// TwinCAT 3 PLC project Core
// Title: Twincat Open Library
// Company: Home
// ProjectVersion: 1.0.0.4
// ProgramVersion: 3.1.4026.17
// libraries:
//   Tc2_Standard, * (Beckhoff Automation GmbH)
//   Tc2_System, * (Beckhoff Automation GmbH)
//   Tc3_Module, * (Beckhoff Automation GmbH)
// project tree:
//   Modules/Common/ E_Requester.TcDUT (not stored), E_RpcMethodResponse.TcDUT, F_ValidateRequester.TcPOU (not stored)
//   Modules/Pneumatics/TwoPosActuator/ E_TwoPosActuator_Fault.TcDUT (not stored), E_TwoPosActuator_State.TcDUT (not stored), FB_TwoPosActuator.TcPOU, ST_TwoPosActuator_Cfg.TcDUT (not stored), ST_TwoPosActuator_IO.TcDUT (not stored), ST_TwoPosActuator_Sts.TcDUT (not stored)
//   Modules/Interlocks/ FB_Interlock.TcPOU (not stored), ST_Interlock_Config.TcDUT (not stored), ST_Interlock_Status.TcDUT (not stored), ST_Interlock_Faceplate.TcDUT (not stored)
//   Modules/Sequencing/Permissives/ FB_Permissives.TcPOU, ST_Permissive_Config.TcDUT (not stored), ST_Permissive_Status.TcDUT (not stored), ST_Permissive_Faceplate.TcDUT
//   Modules/Sequencing/StateMachine/ E_SM_State.TcDUT, FB_StateMachine.TcPOU, FB_Step.TcPOU, ST_SM_Status.TcDUT, ST_SM_Step.TcDUT
//   / PlcTask.TcTTO (not stored)
// (motion and I/O tree: see PLC project coreexample)
// real-time tasks:
//   TASK PlcTask: cycle T#10ms, priority 20, ADS port 350
//   TASK VISU_TASK: cycle T#200000us, priority 30, ADS port 351
//   TASK IO Task New: cycle T#1ms, priority 1, ADS port 301
// variable links:

// ---- Modules/Common/E_RpcMethodResponse.TcDUT
{attribute 'qualified_only'}
{attribute 'strict'}
{attribute 'to_string'}
TYPE E_RpcMethodResponse :
(
    // Success (0)
    ACCEPTED := 0,
    
    // Source / Authorization (10-19)
    REJECTED_SOURCE_NOT_ALLOWED := 11,
    
    // State rejection (20-29)
    REJECTED_WRONG_STATE := 20,
    REJECTED_FAULTED := 21,
    REJECTED_ALREADY_AT_TARGET := 23,
    
    // Parameter / Config (30-39)
    REJECTED_INVALID_PARAMETER := 30,
    REJECTED_BYPASS_NOT_ALLOWED := 31,
    
    // Permissive / Interlock (50-59)
    REJECTED_PERMISSIVE_NOT_MET := 50,
    REJECTED_INTERLOCKED := 51,
    
    // Default (100)
    REJECTED_UNKNOWN := 100
);
END_TYPE

// ---- Modules/Sequencing/Permissives/ST_Permissive_Faceplate.TcDUT
(*
Permissive Faceplate Structure
==============================
Individual permissive bit information for HMI faceplate display
*)
{attribute 'OPC.UA.DA' := '1'}
{attribute 'OPC.UA.DA.Access' := '1'}
{attribute 'OPC.UA.DA.StructuredType' := '1'}
TYPE ST_Permissive_Faceplate :
STRUCT
	{attribute 'OPC.UA.DA.Description' := 'Human readable name of the permissive'}
	name : STRING(50);
	{attribute 'OPC.UA.DA.Description' := 'Real-time status of this permissive bit (TRUE=good, FALSE=bad)'}
	stsOK : BOOL;
	{attribute 'OPC.UA.DA.Description' := 'TRUE if this bit is actively mapped via MapInput'}
	stsMapped : BOOL;
	{attribute 'OPC.UA.DA.Description' := 'TRUE if this bit is currently bypassed'}
	stsBypassed : BOOL;
	{attribute 'OPC.UA.DA.Description' := 'TRUE if this bit is configured as bypassable'}
	cfgBypassable : BOOL;
END_STRUCT
END_TYPE

// ---- Modules/Sequencing/StateMachine/E_SM_State.TcDUT
{attribute 'qualified_only'}
{attribute 'strict'}
{attribute 'to_string'}
TYPE E_SM_State :
(
    IDLE        := 0,
    RUNNING     := 1,
    STOPPING    := 2,
    HOMING      := 4,
    ABORTING    := 8,
    HOMED       := 16,
    STOPPED     := 32,
    ABORTED     := 64,
    COMPLETE    := 128,
    PAUSING     := 256,
    PAUSED      := 512,
    PROCEEDING  := 1024
);
END_TYPE

// ---- Modules/Sequencing/StateMachine/ST_SM_Status.TcDUT
TYPE ST_SM_Status :
STRUCT
    // Current state (enum with to_string for HMI)
    State : E_SM_State := E_SM_State.STOPPED;
    LastState : E_SM_State := E_SM_State.STOPPED;
    
    // Derived state categories
    ActiveState : BOOL;
    WaitingState : BOOL;
    
    // Computed status
    Faulted : BOOL;
    SubmoduleFaulted : BOOL;
    Blocked : BOOL;
    Starved : BOOL;
    
    // Permission-derived readiness
    ReadyToHome : BOOL;
    ReadyToStart : BOOL;
    ReadyToProceed : BOOL;
    
    // Auto-run tracking
    AutoStartRequest : BOOL;
    AutoCycleRequest : BOOL;
END_STRUCT
END_TYPE

// ---- Modules/Sequencing/StateMachine/ST_SM_Step.TcDUT
(*
Active step snapshot published by FB_StateMachine.
FB_Step writes the name and permissives into here while it is the
active step. Number, next target, and timer are owned by the state
machine itself.
*)
{attribute 'OPC.UA.DA' := '1'}
{attribute 'OPC.UA.DA.Access' := '1'}
{attribute 'OPC.UA.DA.StructuredType' := '1'}
TYPE ST_SM_Step :
STRUCT
    {attribute 'OPC.UA.DA.Description' := 'Active step number'}
    Current : DINT;

    {attribute 'OPC.UA.DA.Description' := 'Active step name (published by FB_Step)'}
    Name : STRING(40);

    {attribute 'OPC.UA.DA.Description' := 'Step the state machine will transition to next'}
    Next : DINT;

    {attribute 'OPC.UA.DA.Description' := 'Seconds spent in the active step'}
    TimerSeconds : REAL;

    {attribute 'OPC.UA.DA.Description' := 'Config of the active step permissives'}
    PermCfg : ST_Permissive_Config;

    {attribute 'OPC.UA.DA.Description' := 'Status of the active step permissives'}
    PermStatus : ST_Permissive_Status;
END_STRUCT
END_TYPE

// ---- Modules/Pneumatics/TwoPosActuator/FB_TwoPosActuator.TcPOU
{attribute 'OPC.UA.DA' := '1'}
FUNCTION_BLOCK FB_TwoPosActuator
VAR_INPUT
    {attribute 'OPC.UA.DA' := '0'}
    EnableIn : BOOL := TRUE;
    
    // Configuration
    {attribute 'OPC.UA.DA' := '1'}
    {attribute 'OPC.UA.DA.Access' := '1'}
    cfg : ST_TwoPosActuator_Cfg;
END_VAR

VAR_OUTPUT
    {attribute 'OPC.UA.DA' := '0'}
    EnableOut : BOOL;
    {attribute 'OPC.UA.DA' := '1'}
    {attribute 'OPC.UA.DA.Access' := '1'}
    sts : ST_TwoPosActuator_Sts;
END_VAR

VAR_IN_OUT
    {attribute 'OPC.UA.DA' := '0'}
    IO : ST_TwoPosActuator_IO;
END_VAR

VAR
    // Composed modules - permissive handlers (visible on OPC)
    advancePermissives : FB_Permissives;
    retractPermissives : FB_Permissives;
    
    // Internal state machine
    {attribute 'OPC.UA.DA' := '0'}
    currentState : E_TwoPosActuator_State := E_TwoPosActuator_State.Undefined;
    {attribute 'OPC.UA.DA' := '0'}
    previousState : E_TwoPosActuator_State;
    
    // Timers for motion
    {attribute 'OPC.UA.DA' := '0'}
    advanceTimer : TON;
    {attribute 'OPC.UA.DA' := '0'}
    retractTimer : TON;
    
    // Edge detection
    {attribute 'OPC.UA.DA' := '0'}
    rTrigAdvanced : R_TRIG;
    {attribute 'OPC.UA.DA' := '0'}
    rTrigRetracted : R_TRIG;
    
    // Internal flags
    {attribute 'OPC.UA.DA' := '0'}
    bothFeedbackActive : BOOL;
    
    // Fault handling
    {attribute 'OPC.UA.DA' := '0'}
    faultLatched : BOOL;
    {attribute 'OPC.UA.DA' := '0'}
    lastFault : E_TwoPosActuator_Fault;
    {attribute 'OPC.UA.DA' := '0'}
    bSourceLockedToProg : BOOL;
END_VAR

//-----------------------------------------------------------------------------
// Main Implementation - FB_TwoPosActuator
// Cyclic monitoring only. All commands issued via methods.
//-----------------------------------------------------------------------------
EnableOut := EnableIn;

IF EnableIn THEN
    
    //-------------------------------------------------------------------------
    // Permissive Evaluation
    //-------------------------------------------------------------------------
    advancePermissives();
    retractPermissives();
    
    //-------------------------------------------------------------------------
    // Feedback Analysis
    //-------------------------------------------------------------------------
    bothFeedbackActive := IO.inFbkAdvanced AND IO.inFbkRetracted;
    
    //-------------------------------------------------------------------------
    // State Machine - Cyclic Monitoring
    // Methods set currentState and IO; body monitors for completion/faults.
    //-------------------------------------------------------------------------
    previousState := currentState;
    
    CASE currentState OF
        
        E_TwoPosActuator_State.Undefined:
            IO.outValveAdvance := FALSE;
            IO.outValveRetract := FALSE;
            
            IF bothFeedbackActive THEN
                currentState := E_TwoPosActuator_State.Fault;
                sts.faultCode := E_TwoPosActuator_Fault.BothFeedbackOn;
                faultLatched := TRUE;
            ELSIF IO.inFbkAdvanced AND NOT IO.inFbkRetracted THEN
                currentState := E_TwoPosActuator_State.Advanced;
            ELSIF IO.inFbkRetracted AND NOT IO.inFbkAdvanced THEN
                currentState := E_TwoPosActuator_State.Retracted;
            END_IF;
        
        E_TwoPosActuator_State.Retracted:
            IF cfg.cfgHoldAtRetracted THEN
                IO.outValveRetract := TRUE;
            ELSE
                IO.outValveRetract := FALSE;
            END_IF;
            IO.outValveAdvance := FALSE;
            
            IF bothFeedbackActive THEN
                currentState := E_TwoPosActuator_State.Fault;
                sts.faultCode := E_TwoPosActuator_Fault.BothFeedbackOn;
                faultLatched := TRUE;
            ELSIF NOT IO.inFbkRetracted THEN
                currentState := E_TwoPosActuator_State.Fault;
                sts.faultCode := E_TwoPosActuator_Fault.UndefinedState;
                faultLatched := TRUE;
            END_IF;
        
        E_TwoPosActuator_State.Advancing:
            IO.outValveAdvance := TRUE;
            IO.outValveRetract := FALSE;
            advanceTimer(IN := TRUE, PT := DINT_TO_TIME(cfg.cfgAdvTimeoutS * 1000));
            
            IF IO.inFbkAdvanced AND NOT IO.inFbkRetracted THEN
                currentState := E_TwoPosActuator_State.Advanced;
                advanceTimer(IN := FALSE);
            ELSIF advanceTimer.Q THEN
                currentState := E_TwoPosActuator_State.Fault;
                sts.faultCode := E_TwoPosActuator_Fault.AdvanceTimeout;
                faultLatched := TRUE;
                advanceTimer(IN := FALSE);
            ELSIF bothFeedbackActive THEN
                currentState := E_TwoPosActuator_State.Fault;
                sts.faultCode := E_TwoPosActuator_Fault.BothFeedbackOn;
                faultLatched := TRUE;
                advanceTimer(IN := FALSE);
            ELSIF NOT advancePermissives.sts.bOK THEN
                currentState := E_TwoPosActuator_State.Fault;
                sts.faultCode := E_TwoPosActuator_Fault.PermissivesNotOK;
                faultLatched := TRUE;
                advanceTimer(IN := FALSE);
            END_IF;
        
        E_TwoPosActuator_State.Advanced:
            IF cfg.cfgHoldAtAdvanced THEN
                IO.outValveAdvance := TRUE;
            ELSE
                IO.outValveAdvance := FALSE;
            END_IF;
            IO.outValveRetract := FALSE;
            
            IF bothFeedbackActive THEN
                currentState := E_TwoPosActuator_State.Fault;
                sts.faultCode := E_TwoPosActuator_Fault.BothFeedbackOn;
                faultLatched := TRUE;
            ELSIF NOT IO.inFbkAdvanced THEN
                currentState := E_TwoPosActuator_State.Fault;
                sts.faultCode := E_TwoPosActuator_Fault.UndefinedState;
                faultLatched := TRUE;
            END_IF;
        
        E_TwoPosActuator_State.Retracting:
            IO.outValveRetract := TRUE;
            IO.outValveAdvance := FALSE;
            retractTimer(IN := TRUE, PT := DINT_TO_TIME(cfg.cfgRetTimeoutS * 1000));
            
            IF IO.inFbkRetracted AND NOT IO.inFbkAdvanced THEN
                currentState := E_TwoPosActuator_State.Retracted;
                retractTimer(IN := FALSE);
            ELSIF retractTimer.Q THEN
                currentState := E_TwoPosActuator_State.Fault;
                sts.faultCode := E_TwoPosActuator_Fault.RetractTimeout;
                faultLatched := TRUE;
                retractTimer(IN := FALSE);
            ELSIF bothFeedbackActive THEN
                currentState := E_TwoPosActuator_State.Fault;
                sts.faultCode := E_TwoPosActuator_Fault.BothFeedbackOn;
                faultLatched := TRUE;
                retractTimer(IN := FALSE);
            ELSIF NOT retractPermissives.sts.bOK THEN
                currentState := E_TwoPosActuator_State.Fault;
                sts.faultCode := E_TwoPosActuator_Fault.PermissivesNotOK;
                faultLatched := TRUE;
                retractTimer(IN := FALSE);
            END_IF;
        
        E_TwoPosActuator_State.Fault:
            IO.outValveAdvance := FALSE;
            IO.outValveRetract := FALSE;
            advanceTimer(IN := FALSE);
            retractTimer(IN := FALSE);
    END_CASE;
    
    //-------------------------------------------------------------------------
    // Status Output Generation
    //-------------------------------------------------------------------------
    sts.state := currentState;
    sts.stsAdvanced := (currentState = E_TwoPosActuator_State.Advanced);
    sts.stsRetracted := (currentState = E_TwoPosActuator_State.Retracted);
    sts.stsMoving := (currentState = E_TwoPosActuator_State.Advancing) OR 
                     (currentState = E_TwoPosActuator_State.Retracting);
    sts.stsFaulted := (currentState = E_TwoPosActuator_State.Fault) OR faultLatched;
    sts.lastFaultCode := lastFault;
    
    rTrigAdvanced(CLK := sts.stsAdvanced);
    sts.osAdvanced := rTrigAdvanced.Q;
    
    rTrigRetracted(CLK := sts.stsRetracted);
    sts.osRetracted := rTrigRetracted.Q;
    
    //-------------------------------------------------------------------------
    // String Generation for OPC/HMI
    //-------------------------------------------------------------------------
    CASE currentState OF
        E_TwoPosActuator_State.Undefined:   sts.stateString := 'Undefined';
        E_TwoPosActuator_State.Retracted:   sts.stateString := 'Retracted';
        E_TwoPosActuator_State.Advancing:   sts.stateString := 'Advancing';
        E_TwoPosActuator_State.Advanced:    sts.stateString := 'Advanced';
        E_TwoPosActuator_State.Retracting:  sts.stateString := 'Retracting';
        E_TwoPosActuator_State.Fault:       sts.stateString := 'Fault';
    ELSE
        sts.stateString := 'Unknown';
    END_CASE;
    
    CASE sts.faultCode OF
        E_TwoPosActuator_Fault.None:               sts.faultString := 'No Fault';
        E_TwoPosActuator_Fault.AdvanceTimeout:      sts.faultString := 'Advance Timeout';
        E_TwoPosActuator_Fault.RetractTimeout:      sts.faultString := 'Retract Timeout';
        E_TwoPosActuator_Fault.BothFeedbackOn:      sts.faultString := 'Both Feedbacks Active';
        E_TwoPosActuator_Fault.UndefinedState:      sts.faultString := 'Position Undefined';
        E_TwoPosActuator_Fault.PermissivesNotOK:    sts.faultString := 'Permissives Not OK';
        E_TwoPosActuator_Fault.ConflictingCommands:  sts.faultString := 'Conflicting Commands';
        E_TwoPosActuator_Fault.NoFeedback:          sts.faultString := 'No Position Feedback';
    ELSE
        sts.faultString := 'Unknown Fault';
    END_CASE;
    
    CASE sts.lastFaultCode OF
        E_TwoPosActuator_Fault.None:               sts.lastFaultString := 'No Previous Fault';
        E_TwoPosActuator_Fault.AdvanceTimeout:      sts.lastFaultString := 'Last: Advance Timeout';
        E_TwoPosActuator_Fault.RetractTimeout:      sts.lastFaultString := 'Last: Retract Timeout';
        E_TwoPosActuator_Fault.BothFeedbackOn:      sts.lastFaultString := 'Last: Both Feedbacks Active';
        E_TwoPosActuator_Fault.UndefinedState:      sts.lastFaultString := 'Last: Position Undefined';
        E_TwoPosActuator_Fault.PermissivesNotOK:    sts.lastFaultString := 'Last: Permissives Not OK';
        E_TwoPosActuator_Fault.ConflictingCommands:  sts.lastFaultString := 'Last: Conflicting Commands';
        E_TwoPosActuator_Fault.NoFeedback:          sts.lastFaultString := 'Last: No Position Feedback';
    ELSE
        sts.lastFaultString := 'Last: Unknown Fault';
    END_CASE;
    
ELSE
    IO.outValveAdvance := FALSE;
    IO.outValveRetract := FALSE;
    advanceTimer(IN := FALSE);
    retractTimer(IN := FALSE);
END_IF;

{attribute 'TcRpcEnable' := '1'}
METHOD PUBLIC Advance : E_RpcMethodResponse
VAR_INPUT
    eRequester : E_Requester := E_Requester.PROG;
END_VAR
// 1. Source + fault validation
Advance := F_ValidateRequester(eRequester, bSourceLockedToProg, faultLatched, FALSE, FALSE);
IF Advance <> E_RpcMethodResponse.ACCEPTED THEN RETURN; END_IF;

// 2. State check — must not already be advanced or advancing
IF currentState = E_TwoPosActuator_State.Advanced OR currentState = E_TwoPosActuator_State.Advancing THEN
    Advance := E_RpcMethodResponse.REJECTED_ALREADY_AT_TARGET;
    RETURN;
END_IF;

// 3. Permissive check
IF NOT advancePermissives.sts.bOK THEN
    Advance := E_RpcMethodResponse.REJECTED_PERMISSIVE_NOT_MET;
    RETURN;
END_IF;

// 4. Execute — set state, body handles the rest
currentState := E_TwoPosActuator_State.Advancing;
advanceTimer(IN := FALSE);
Advance := E_RpcMethodResponse.ACCEPTED;
END_METHOD

{attribute 'TcRpcEnable' := '1'}
METHOD PUBLIC Retract : E_RpcMethodResponse
VAR_INPUT
    eRequester : E_Requester := E_Requester.PROG;
END_VAR
// 1. Source + fault validation
Retract := F_ValidateRequester(eRequester, bSourceLockedToProg, faultLatched, FALSE, FALSE);
IF Retract <> E_RpcMethodResponse.ACCEPTED THEN RETURN; END_IF;

// 2. State check — must not already be retracted or retracting
IF currentState = E_TwoPosActuator_State.Retracted OR currentState = E_TwoPosActuator_State.Retracting THEN
    Retract := E_RpcMethodResponse.REJECTED_ALREADY_AT_TARGET;
    RETURN;
END_IF;

// 3. Permissive check
IF NOT retractPermissives.sts.bOK THEN
    Retract := E_RpcMethodResponse.REJECTED_PERMISSIVE_NOT_MET;
    RETURN;
END_IF;

// 4. Execute — set state, body handles the rest
currentState := E_TwoPosActuator_State.Retracting;
retractTimer(IN := FALSE);
Retract := E_RpcMethodResponse.ACCEPTED;
END_METHOD

{attribute 'TcRpcEnable' := '1'}
METHOD PUBLIC AllOff : E_RpcMethodResponse
VAR_INPUT
    eRequester : E_Requester := E_Requester.PROG;
END_VAR
// AllOff is always accepted — safety command
AllOff := F_ValidateRequester(eRequester, bSourceLockedToProg, faultLatched, FALSE, TRUE);
IF AllOff <> E_RpcMethodResponse.ACCEPTED THEN RETURN; END_IF;

IO.outValveAdvance := FALSE;
IO.outValveRetract := FALSE;
advanceTimer(IN := FALSE);
retractTimer(IN := FALSE);
currentState := E_TwoPosActuator_State.Undefined;
AllOff := E_RpcMethodResponse.ACCEPTED;
END_METHOD

{attribute 'TcRpcEnable' := '1'}
METHOD PUBLIC Reset : E_RpcMethodResponse
VAR_INPUT
    eRequester : E_Requester := E_Requester.PROG;
END_VAR
// 1. Source validation — allow when faulted
Reset := F_ValidateRequester(eRequester, bSourceLockedToProg, faultLatched, TRUE, FALSE);
IF Reset <> E_RpcMethodResponse.ACCEPTED THEN RETURN; END_IF;

// 2. Must be in fault state
IF currentState <> E_TwoPosActuator_State.Fault THEN
    Reset := E_RpcMethodResponse.REJECTED_WRONG_STATE;
    RETURN;
END_IF;

// 3. Execute — clear fault and go to Undefined for re-evaluation
lastFault := sts.faultCode;
faultLatched := FALSE;
sts.faultCode := E_TwoPosActuator_Fault.None;
currentState := E_TwoPosActuator_State.Undefined;
IO.outValveAdvance := FALSE;
IO.outValveRetract := FALSE;
Reset := E_RpcMethodResponse.ACCEPTED;
END_METHOD

{attribute 'TcRpcEnable' := '1'}
METHOD PUBLIC LockSource : E_RpcMethodResponse
VAR_INPUT
    bLock : BOOL;
END_VAR
bSourceLockedToProg := bLock;
LockSource := E_RpcMethodResponse.ACCEPTED;
END_METHOD

END_FUNCTION_BLOCK

// ---- Modules/Sequencing/Permissives/FB_Permissives.TcPOU
(*
PERMISSIVE - Operational Enabling Function Block
================================================
Philosophy: 	Allows a change in state when all conditions are met
Behavior: 		Follows real-time conditions, no latching, can be bypassed for maintenance
Logic: 			Mapped bits: 1 = good, 0 = bad. Unmapped bits are automatically good (1)
				sts.bOK = TRUE when ALL active permissive bits are good (or bypassed)
				Non-latching - immediate response to condition changes
Mapping:		Use MapInput method to assign boolean signals to specific bits (0..63)
				Unmapped bits automatically return to good state after timeout
*)
{attribute 'OPC.UA.DA' := '1'}
FUNCTION_BLOCK PUBLIC FB_Permissives
VAR_INPUT
	{attribute 'OPC.UA.DA' := '1'}
	{attribute 'OPC.UA.DA.Access' := '1'}
	cfg : ST_Permissive_Config;
END_VAR
VAR_OUTPUT
	{attribute 'OPC.UA.DA' := '1'}
	{attribute 'OPC.UA.DA.Access' := '1'}
	sts : ST_Permissive_Status;
END_VAR
VAR
	{attribute 'OPC.UA.DA' := '0'}
	_permissiveBits : ULINT := 16#FFFFFFFFFFFFFFFF;	// Working bits (1=good, 0=bad), default all good
	{attribute 'OPC.UA.DA' := '0'}
	_activeMask : ULINT := 0;							// Tracks which bits are actively mapped
	{attribute 'OPC.UA.DA' := '0'}
	_bypassMask : ULINT := 0;							// Dynamic bypass mask (1=bypassed)
	{attribute 'OPC.UA.DA' := '0'}
	_previousBits : ULINT := 16#FFFFFFFFFFFFFFFF;		// Previous cycle bits for transition detection
	{attribute 'OPC.UA.DA' := '0'}
	_cycleCounter : UDINT := 0;
	{attribute 'OPC.UA.DA' := '0'}
	_lastMappedCycle : ARRAY[0..63] OF UDINT;
	{attribute 'OPC.UA.DA' := '0'}
	_sequenceCounter : UDINT := 0;
	{attribute 'OPC.UA.DA' := '0'}
	MAPPING_TIMEOUT : UDINT := 10;						// Cycles before considering a bit unmapped
END_VAR

// Increment cycle counter
_cycleCounter := _cycleCounter + 1;
IF _cycleCounter = 0 THEN _cycleCounter := 1; END_IF

// Cleanup unmapped bits
CleanupUnmappedBits();

// Detect transitions for first-failure tracking
DetectTransitions();

// Compute permissive status: unmapped bits default good, then apply bypass
sts.nPermissives := (_permissiveBits OR NOT _activeMask) OR _bypassMask;
sts.nBypassMask := _bypassMask;

// Overall OK: all 64 bits good
sts.bOK := sts.nPermissives = 16#FFFFFFFFFFFFFFFF;

// Update faceplates for HMI
UpdateFaceplates();

// Store for next cycle transition detection
_previousBits := _permissiveBits;

METHOD PRIVATE CleanupUnmappedBits
VAR
	i : UDINT;
	bitMask : ULINT;
END_VAR
FOR i := 0 TO 63 DO
	bitMask := SHL(ULINT#1, i);
	IF (_activeMask AND bitMask) <> 0 THEN
		IF (_cycleCounter - _lastMappedCycle[i]) > MAPPING_TIMEOUT THEN
			_activeMask := _activeMask AND NOT bitMask;
			_permissiveBits := _permissiveBits OR bitMask;	// Reset to good
		END_IF
	END_IF
END_FOR;
END_METHOD

METHOD PRIVATE DetectTransitions
VAR
	i : UDINT;
	bitMask : ULINT;
END_VAR
// New failure sequence: transition from all-good to first failure
IF _previousBits = 16#FFFFFFFFFFFFFFFF AND _permissiveBits <> 16#FFFFFFFFFFFFFFFF THEN
	_sequenceCounter := 0;
	sts.nFirstFailureBitIndex := 999;
END_IF

// Detect good-to-bad transitions on active bits
FOR i := 0 TO 63 DO
	bitMask := SHL(ULINT#1, i);
	IF (_activeMask AND bitMask) <> 0 THEN
		// Previous good (1) AND current bad (0) = transition
		IF ((_previousBits AND bitMask) <> 0) AND ((_permissiveBits AND bitMask) = 0) THEN
			_sequenceCounter := _sequenceCounter + 1;
			IF _sequenceCounter = 1 THEN
				sts.nFirstFailureBitIndex := i;
			END_IF
		END_IF
	END_IF
END_FOR;
END_METHOD

(*
Map a boolean input signal to a specific permissive bit (0..63)
Call every cycle for each active permissive condition
*)
METHOD PUBLIC MapInput
VAR_INPUT
	bitIndex : UDINT;
	inputValue : BOOL;
END_VAR
VAR
	bitMask : ULINT;
END_VAR
IF bitIndex > 63 THEN RETURN; END_IF

bitMask := SHL(ULINT#1, bitIndex);
_activeMask := _activeMask OR bitMask;
_lastMappedCycle[bitIndex] := _cycleCounter;

IF inputValue THEN
	_permissiveBits := _permissiveBits OR bitMask;
ELSE
	_permissiveBits := _permissiveBits AND NOT bitMask;
END_IF;
END_METHOD

(*
Reset - Clear all bypass states
Permissives continue to follow real-time conditions (non-latching)
*)
{attribute 'TcRpcEnable':='1'}
METHOD Reset
_bypassMask := 0;
END_METHOD

(*
Set or clear bypass for a specific permissive bit
Only bits configured as bypassable in cfg.nBypassable can be bypassed
Clearing bypass (bEnable := FALSE) is always allowed
*)
{attribute 'TcRpcEnable':='1'}
METHOD PUBLIC SetBypass : E_RpcMethodResponse
VAR_INPUT
	bitIndex : UDINT;
	bEnable : BOOL;
END_VAR
VAR
	bitMask : ULINT;
END_VAR
IF bitIndex > 63 THEN
	SetBypass := E_RpcMethodResponse.REJECTED_INVALID_PARAMETER;
	RETURN;
END_IF

bitMask := SHL(ULINT#1, bitIndex);

// Only check bypassable config when enabling
IF bEnable AND (cfg.nBypassable AND bitMask) = 0 THEN
	SetBypass := E_RpcMethodResponse.REJECTED_BYPASS_NOT_ALLOWED;
	RETURN;
END_IF

IF bEnable THEN
	_bypassMask := _bypassMask OR bitMask;
ELSE
	_bypassMask := _bypassMask AND NOT bitMask;
END_IF

SetBypass := E_RpcMethodResponse.ACCEPTED;
END_METHOD

METHOD PRIVATE UpdateFaceplates
VAR
	i : UDINT;
	bitMask : ULINT;
END_VAR
FOR i := 0 TO 63 DO
	bitMask := SHL(ULINT#1, i);
	sts.aFaceplates[i].name := cfg.aNames[i];
	sts.aFaceplates[i].stsOK := (sts.nPermissives AND bitMask) <> 0;
	sts.aFaceplates[i].stsMapped := (_activeMask AND bitMask) <> 0;
	sts.aFaceplates[i].stsBypassed := (_bypassMask AND bitMask) <> 0;
	sts.aFaceplates[i].cfgBypassable := (cfg.nBypassable AND bitMask) <> 0;
END_FOR;
END_METHOD

END_FUNCTION_BLOCK

// ---- Modules/Sequencing/StateMachine/FB_StateMachine.TcPOU
FUNCTION_BLOCK FB_StateMachine
VAR_INPUT
    EnableIn : BOOL;
    cfgAutoRun : BOOL;
    inpBlockedCondition : DINT;
    inpStarvedCondition : DINT;
    inpSubmoduleFaulted : BOOL;
END_VAR

VAR_OUTPUT
    EnableOut : BOOL;
    Status : ST_SM_Status;
END_VAR

VAR CONSTANT
    HOMING_MIN   : DINT := 1000; HOMING_MAX   : DINT := 1999;
    RUNNING_MIN  : DINT := 3000; RUNNING_MAX  : DINT := 3999;
    STOPPING_MIN : DINT := 2000; STOPPING_MAX : DINT := 2999;
    ABORTING_MIN : DINT := 5000; ABORTING_MAX : DINT := 5999;
    PAUSING_MIN  : DINT := 4000; PAUSING_MAX  : DINT := 4999;
    PROCEEDING_MIN : DINT := 6000; PROCEEDING_MAX : DINT := 6999;
END_VAR

VAR
    // Internal command request flags (set by methods, consumed by body)
    _abortRequested : BOOL;
    _completeStateRequested : BOOL;
    _homeRequested : BOOL;
    _pauseRequested : BOOL;
    _proceedRequested : BOOL;
    _startRequested : BOOL;
    _stopRequested : BOOL;
    _retryActive : BOOL;
    RetryComplete : BOOL;
    
    // Timer
    StepTimer : TON;
    
    // Edge detection
    R_TRIG_1 : R_TRIG;
    R_TRIG_5 : R_TRIG;
    
    // Internal state tracking
    _previousState : E_SM_State;
    PreviousStep : DINT;
    TimerReset : BOOL;
    LsOdd : DINT;
    _returnState : E_SM_State;
    ReturnNextStep : DINT;
    
    // Permission handlers
    permAuto : FB_Permissives;
    permHome : FB_Permissives;
    permProceed : FB_Permissives;
    permStart : FB_Permissives;
    
    // Running interlock (latching - auto-aborts from any active state)
    intlkRunning : FB_Interlock;
    
    // Temp variables
    permIndex : UDINT;
    stepIsZero : BOOL;
    seqDone : BOOL;
    
    // Source control
    bSourceLockedToProg : BOOL;
    
    // Step ownership (internal)
    _nextStep : DINT;
END_VAR


//-----------------------------------------------------------------------------
// Main Implementation
//-----------------------------------------------------------------------------
EnableOut := EnableIn;

// Only execute if enabled
IF EnableIn THEN
    //-------------------------------------------------------------------------
    // Process permissions for different states
    //-------------------------------------------------------------------------
    permHome();
    permStart();
    permProceed();
    permAuto();
    
    intlkRunning();
    
    // Auto-abort if any running interlock trips (e-stop, safety gate, etc.)
    IF NOT intlkRunning.sts.bOK AND
       NOT (Status.State = E_SM_State.STOPPED OR Status.State = E_SM_State.ABORTING) THEN
        _abortRequested := TRUE;
    END_IF;
    
    //-------------------------------------------------------------------------
    // Ready state calculations
    //-------------------------------------------------------------------------
    Status.ReadyToHome := (Status.State = E_SM_State.STOPPED) AND
                          permHome.sts.bOK AND
                          permAuto.sts.bOK;

    Status.ReadyToStart := (Status.State = E_SM_State.READY) AND
                          permStart.sts.bOK AND
                          permAuto.sts.bOK AND
                          NOT Status.AutoStartRequest;

    Status.ReadyToProceed := (Status.State = E_SM_State.PAUSED) AND
                            permProceed.sts.bOK AND
                            permAuto.sts.bOK;

    //-------------------------------------------------------------------------
    // Auto-start request logic
    // AutoCycle fires when we just finished a RUNNING cycle (READY with LastState=RUNNING)
    //-------------------------------------------------------------------------
    Status.AutoStartRequest := _startRequested AND NOT permStart.sts.bOK;
    Status.AutoCycleRequest := cfgAutoRun AND (Status.State = E_SM_State.READY) AND
                              (Status.LastState = E_SM_State.RUNNING) AND NOT permStart.sts.bOK;

    //-------------------------------------------------------------------------
    // Remember last state before change
    //-------------------------------------------------------------------------
    _previousState := Status.State;

    //-------------------------------------------------------------------------
    // Auto-run handling (internal - not from external command)
    //-------------------------------------------------------------------------
    IF cfgAutoRun AND permAuto.sts.bOK AND permStart.sts.bOK AND
       (Status.State = E_SM_State.READY) AND (Status.LastState = E_SM_State.RUNNING) THEN
        _startRequested := TRUE;
    END_IF;
    
    //-------------------------------------------------------------------------
    // Sequence completion inference
    //-------------------------------------------------------------------------
    seqDone := _IsStepInStateRange(
        state := Status.State,
        nStep := Status.Step.Current
    ) AND (_nextStep = 0);

    R_TRIG_5(CLK := seqDone);
    IF R_TRIG_5.Q THEN
        _completeStateRequested := TRUE;
    END_IF;

    //-------------------------------------------------------------------------
    // State Transitions
    //-------------------------------------------------------------------------

    // Homing complete → Ready
    IF _completeStateRequested AND (Status.State = E_SM_State.HOMING) THEN
        _nextStep := 0;
        Status.State := E_SM_State.READY;
        _completeStateRequested := FALSE;
    END_IF;

    // Running complete → Ready (LastState will be RUNNING so AutoCycle can detect a just-finished cycle)
    IF _completeStateRequested AND (Status.State = E_SM_State.RUNNING) THEN
        _nextStep := 0;
        Status.State := E_SM_State.READY;
        _completeStateRequested := FALSE;
    END_IF;

    // Running + Stop → Stopping
    IF _stopRequested AND (Status.State = E_SM_State.RUNNING) THEN
        Status.State := E_SM_State.STOPPING;
    END_IF;

    // Stopping complete → Stopped
    IF _completeStateRequested AND (Status.State = E_SM_State.STOPPING) THEN
        _nextStep := 0;
        Status.State := E_SM_State.STOPPED;
        _completeStateRequested := FALSE;
    END_IF;

    // Aborting complete → Stopped (Status.Faulted remains indicated via LastState = ABORTING)
    IF _completeStateRequested AND (Status.State = E_SM_State.ABORTING) THEN
        _nextStep := 0;
        Status.State := E_SM_State.STOPPED;
        _completeStateRequested := FALSE;
    END_IF;

    // Running + Pause → Pausing (save context for Proceed)
    IF _pauseRequested AND (Status.State = E_SM_State.RUNNING) THEN
        _returnState := Status.State;
        ReturnNextStep := Status.Step.Current;  // resume re-enters same step
        Status.State := E_SM_State.PAUSING;
        _nextStep := 0;
    END_IF;

    // Pausing complete → Paused
    IF _completeStateRequested AND (Status.State = E_SM_State.PAUSING) THEN
        _nextStep := 0;
        Status.State := E_SM_State.PAUSED;
        _completeStateRequested := FALSE;
    END_IF;

    // Proceeding complete → return to state before pause, re-enter the paused step
    IF _completeStateRequested AND (Status.State = E_SM_State.PROCEEDING) THEN
        _nextStep := ReturnNextStep;
        Status.State := _returnState;
        _completeStateRequested := FALSE;
    END_IF;

    // Ready + Start → Running
    IF (_startRequested OR
        (Status.AutoStartRequest AND permStart.sts.bOK AND permAuto.sts.bOK)) AND
        (Status.State = E_SM_State.READY) THEN
        _nextStep := 0;
        Status.State := E_SM_State.RUNNING;
        _startRequested := FALSE;
    END_IF;

    // Ready + Stop → Stopped (no sequence needed, machine is already quiescent)
    IF _stopRequested AND (Status.State = E_SM_State.READY) THEN
        _nextStep := 0;
        Status.State := E_SM_State.STOPPED;
    END_IF;

    // Stopped + Home → Homing
    IF _homeRequested AND (Status.State = E_SM_State.STOPPED) THEN
        _nextStep := 0;
        Status.State := E_SM_State.HOMING;
    END_IF;

    // Paused + Proceed → Proceeding
    IF _proceedRequested AND (Status.State = E_SM_State.PAUSED) THEN
        _nextStep := 0;
        Status.State := E_SM_State.PROCEEDING;
    END_IF;

    // Abort from any state except Stopped / Aborting
    IF _abortRequested AND NOT (Status.State = E_SM_State.STOPPED OR Status.State = E_SM_State.ABORTING) THEN
        _nextStep := 0;
        Status.State := E_SM_State.ABORTING;
    END_IF;
    
    //-------------------------------------------------------------------------
    // Track state changes
    //-------------------------------------------------------------------------
    IF Status.State <> _previousState THEN
        Status.LastState := _previousState;
    END_IF;
    
    //-------------------------------------------------------------------------
    // Derived status flags
    //-------------------------------------------------------------------------
    Status.WaitingState := (Status.State = E_SM_State.STOPPED) OR (Status.State = E_SM_State.READY) OR
                           (Status.State = E_SM_State.PAUSED);
    Status.ActiveState  := (Status.State = E_SM_State.HOMING) OR (Status.State = E_SM_State.RUNNING) OR
                           (Status.State = E_SM_State.STOPPING) OR (Status.State = E_SM_State.PAUSING) OR
                           (Status.State = E_SM_State.PROCEEDING) OR (Status.State = E_SM_State.ABORTING);

    //-------------------------------------------------------------------------
    // Step and timer management
    //-------------------------------------------------------------------------
    
    // Reset timer and clear step name when transitioning to step 0
    stepIsZero := (Status.Step.Current = 0);
    R_TRIG_1(CLK := stepIsZero);
    IF R_TRIG_1.Q THEN
        Status.Step.Name := '';
        _ClearStepPermissives();
        TimerReset := TRUE;
        StepTimer(IN := FALSE, PT := T#99H);
        Status.Step.TimerSeconds := 0.0;
    END_IF;
    
    // Auto-initialize first step when entering an active state
    IF Status.Step.Current = 0 AND Status.ActiveState THEN
        _nextStep := _GetFirstStepForState(state := Status.State);
    END_IF;
    
    // Detect step change and update
    IF Status.Step.Current <> _nextStep THEN
        PreviousStep := Status.Step.Current;
        Status.Step.Current := _nextStep;
        TimerReset := TRUE;
        StepTimer(IN := FALSE, PT := T#99H);
        Status.Step.TimerSeconds := 0.0;
    END_IF;
    
    Status.Step.Next := _nextStep;
    
    // Step timer logic
    IF NOT (Status.State = E_SM_State.PAUSED) OR ((Status.State = E_SM_State.PAUSED) AND _completeStateRequested) THEN
        IF TimerReset THEN
            StepTimer(IN := FALSE, PT := T#99H);
            Status.Step.TimerSeconds := 0.0;
            TimerReset := FALSE;
        ELSE
            StepTimer(IN := TRUE, PT := T#99H);
            Status.Step.TimerSeconds := UDINT_TO_REAL(TIME_TO_UDINT(StepTimer.ET)) / 1000.0;
        END_IF;
    ELSE
        StepTimer(IN := FALSE, PT := T#99H);
    END_IF;
    
    //-------------------------------------------------------------------------
    // Fault detection
    //-------------------------------------------------------------------------
    LsOdd := Status.Step.Current MOD 2;
    Status.Faulted := LsOdd <> 0;
    Status.SubmoduleFaulted := inpSubmoduleFaulted;
    
    //-------------------------------------------------------------------------
    // Retry logic
    //-------------------------------------------------------------------------
    IF RetryComplete THEN
        _retryActive := FALSE;
        RetryComplete := FALSE;
    END_IF;
    
    IF _retryActive THEN
        RetryComplete := TRUE;
    END_IF;
    
    IF _retryActive AND Status.Faulted THEN
        // Roll back to previous (even, non-faulted) step to re-enter it
        _nextStep := Status.Step.Current - 1;
    END_IF;
    
    //-------------------------------------------------------------------------
    // OEE condition codes (Blocked / Starved)
    //-------------------------------------------------------------------------
    IF inpBlockedCondition = 0 THEN
        Status.BlockedCondition := 0;
    END_IF;
    
    IF inpBlockedCondition <> 0 AND
       (Status.State = E_SM_State.RUNNING OR Status.State = E_SM_State.STOPPING OR
        Status.State = E_SM_State.READY) THEN
        Status.BlockedCondition := inpBlockedCondition;
        inpBlockedCondition := 0;
    END_IF;
    
    IF inpStarvedCondition = 0 THEN
        Status.StarvedCondition := 0;
    END_IF;
    
    IF inpStarvedCondition <> 0 AND
       (Status.State = E_SM_State.RUNNING OR Status.State = E_SM_State.STOPPING OR
        Status.State = E_SM_State.READY) THEN
        Status.StarvedCondition := inpStarvedCondition;
        inpStarvedCondition := 0;
    END_IF;
    
ELSE
    // Reset command requests when disabled
    _startRequested := FALSE;
    _stopRequested := FALSE;
    _homeRequested := FALSE;
    _abortRequested := FALSE;
    _pauseRequested := FALSE;
    _proceedRequested := FALSE;
    _completeStateRequested := FALSE;
    Status.Step.Name := '';
        _ClearStepPermissives();
END_IF;

METHOD PRIVATE _ClearStepPermissives
Status.Step.PermCfg.nBypassable := 0;
Status.Step.PermStatus.bOK := FALSE;
Status.Step.PermStatus.nPermissives := 0;
Status.Step.PermStatus.nBypassMask := 0;
Status.Step.PermStatus.nFirstFailureBitIndex := 999;

FOR permIndex := 0 TO 63 DO
        Status.Step.PermCfg.aNames[permIndex] := '';
        Status.Step.PermStatus.aFaceplates[permIndex].name := '';
        Status.Step.PermStatus.aFaceplates[permIndex].stsOK := FALSE;
        Status.Step.PermStatus.aFaceplates[permIndex].stsMapped := FALSE;
        Status.Step.PermStatus.aFaceplates[permIndex].stsBypassed := FALSE;
        Status.Step.PermStatus.aFaceplates[permIndex].cfgBypassable := FALSE;
END_FOR;
END_METHOD

METHOD PRIVATE _GetFirstStepForState : DINT
VAR_INPUT
        state : E_SM_State;
END_VAR
CASE state OF
        E_SM_State.HOMING:     _GetFirstStepForState := HOMING_MIN;
        E_SM_State.RUNNING:    _GetFirstStepForState := RUNNING_MIN;
        E_SM_State.STOPPING:   _GetFirstStepForState := STOPPING_MIN;
        E_SM_State.ABORTING:   _GetFirstStepForState := ABORTING_MIN;
        E_SM_State.PAUSING:    _GetFirstStepForState := PAUSING_MIN;
        E_SM_State.PROCEEDING: _GetFirstStepForState := PROCEEDING_MIN;
ELSE
        _GetFirstStepForState := 0;
END_CASE;
END_METHOD

METHOD PRIVATE _GetLastStepForState : DINT
VAR_INPUT
        state : E_SM_State;
END_VAR
CASE state OF
        E_SM_State.HOMING:     _GetLastStepForState := HOMING_MAX;
        E_SM_State.RUNNING:    _GetLastStepForState := RUNNING_MAX;
        E_SM_State.STOPPING:   _GetLastStepForState := STOPPING_MAX;
        E_SM_State.ABORTING:   _GetLastStepForState := ABORTING_MAX;
        E_SM_State.PAUSING:    _GetLastStepForState := PAUSING_MAX;
        E_SM_State.PROCEEDING: _GetLastStepForState := PROCEEDING_MAX;
ELSE
        _GetLastStepForState := 0;
END_CASE;
END_METHOD

METHOD PRIVATE _IsStepInStateRange : BOOL
VAR_INPUT
        state : E_SM_State;
        nStep : DINT;
END_VAR
_IsStepInStateRange := (nStep >= _GetFirstStepForState(state := state)) AND
                                             (nStep <= _GetLastStepForState(state := state));
END_METHOD

{attribute 'TcRpcEnable' := '1'}
METHOD Abort : E_RpcMethodResponse
VAR_INPUT
    eRequester : E_Requester := E_Requester.PROG;
END_VAR
// Safety command - skip source check, skip fault check
IF Status.State = E_SM_State.STOPPED OR Status.State = E_SM_State.ABORTING THEN
    Abort := E_RpcMethodResponse.REJECTED_WRONG_STATE;
    RETURN;
END_IF;

// Execute - clear other requests, set abort
_startRequested := FALSE;
_stopRequested := FALSE;
_homeRequested := FALSE;
_pauseRequested := FALSE;
_proceedRequested := FALSE;
_completeStateRequested := FALSE;
_abortRequested := TRUE;
Abort := E_RpcMethodResponse.ACCEPTED;
END_METHOD

{attribute 'TcRpcEnable' := '1'}
METHOD Home : E_RpcMethodResponse
VAR_INPUT
    eRequester : E_Requester := E_Requester.PROG;
END_VAR
// Common validation
Home := F_ValidateRequester(eRequester, bSourceLockedToProg, Status.Faulted, FALSE, FALSE);
IF Home <> E_RpcMethodResponse.ACCEPTED THEN RETURN; END_IF;

// State check
IF NOT (Status.State = E_SM_State.STOPPED) THEN
    Home := E_RpcMethodResponse.REJECTED_WRONG_STATE;
    RETURN;
END_IF;

// Permission check (Home-specific)
IF NOT permHome.sts.bOK THEN
    Home := E_RpcMethodResponse.REJECTED_PERMISSIVE_NOT_MET;
    RETURN;
END_IF;

// Permission check (global auto permissives)
IF NOT permAuto.sts.bOK THEN
    Home := E_RpcMethodResponse.REJECTED_PERMISSIVE_NOT_MET;
    RETURN;
END_IF;

// Execute
_abortRequested := FALSE;
_pauseRequested := FALSE;
_proceedRequested := FALSE;
_startRequested := FALSE;
_stopRequested := FALSE;
_completeStateRequested := FALSE;
_homeRequested := TRUE;
Home := E_RpcMethodResponse.ACCEPTED;
END_METHOD

METHOD LockSource
VAR_INPUT
    bLock : BOOL;
END_VAR
bSourceLockedToProg := bLock;
END_METHOD

{attribute 'TcRpcEnable' := '1'}
METHOD Pause : E_RpcMethodResponse
VAR_INPUT
    eRequester : E_Requester := E_Requester.PROG;
END_VAR
// Common validation
Pause := F_ValidateRequester(eRequester, bSourceLockedToProg, Status.Faulted, FALSE, FALSE);
IF Pause <> E_RpcMethodResponse.ACCEPTED THEN RETURN; END_IF;

// State check
IF NOT (Status.State = E_SM_State.RUNNING) THEN
    Pause := E_RpcMethodResponse.REJECTED_WRONG_STATE;
    RETURN;
END_IF;

// Execute
_abortRequested := FALSE;
_homeRequested := FALSE;
_proceedRequested := FALSE;
_startRequested := FALSE;
_stopRequested := FALSE;
_completeStateRequested := FALSE;
_pauseRequested := TRUE;
Pause := E_RpcMethodResponse.ACCEPTED;
END_METHOD

{attribute 'TcRpcEnable' := '1'}
METHOD Proceed : E_RpcMethodResponse
VAR_INPUT
    eRequester : E_Requester := E_Requester.PROG;
END_VAR
// Common validation
Proceed := F_ValidateRequester(eRequester, bSourceLockedToProg, Status.Faulted, FALSE, FALSE);
IF Proceed <> E_RpcMethodResponse.ACCEPTED THEN RETURN; END_IF;

// State check
IF NOT (Status.State = E_SM_State.PAUSED) THEN
    Proceed := E_RpcMethodResponse.REJECTED_WRONG_STATE;
    RETURN;
END_IF;

// Permission check (Proceed-specific)
IF NOT permProceed.sts.bOK THEN
    Proceed := E_RpcMethodResponse.REJECTED_PERMISSIVE_NOT_MET;
    RETURN;
END_IF;

// Permission check (global auto permissives)
IF NOT permAuto.sts.bOK THEN
    Proceed := E_RpcMethodResponse.REJECTED_PERMISSIVE_NOT_MET;
    RETURN;
END_IF;

// Execute
_abortRequested := FALSE;
_homeRequested := FALSE;
_pauseRequested := FALSE;
_startRequested := FALSE;
_stopRequested := FALSE;
_completeStateRequested := FALSE;
_proceedRequested := TRUE;
Proceed := E_RpcMethodResponse.ACCEPTED;
END_METHOD

{attribute 'TcRpcEnable' := '1'}
METHOD Retry : E_RpcMethodResponse
VAR_INPUT
    eRequester : E_Requester := E_Requester.PROG;
END_VAR
// Common validation
Retry := F_ValidateRequester(eRequester, bSourceLockedToProg, Status.Faulted, FALSE, FALSE);
IF Retry <> E_RpcMethodResponse.ACCEPTED THEN RETURN; END_IF;

// Execute - set retry directly
_retryActive := TRUE;
Retry := E_RpcMethodResponse.ACCEPTED;
END_METHOD

{attribute 'TcRpcEnable' := '1'}
METHOD Start : E_RpcMethodResponse
VAR_INPUT
    eRequester : E_Requester := E_Requester.PROG;
END_VAR
// Common validation
Start := F_ValidateRequester(eRequester, bSourceLockedToProg, Status.Faulted, FALSE, FALSE);
IF Start <> E_RpcMethodResponse.ACCEPTED THEN RETURN; END_IF;

// State check
IF NOT (Status.State = E_SM_State.READY) THEN
    Start := E_RpcMethodResponse.REJECTED_WRONG_STATE;
    RETURN;
END_IF;

// Permission check (Start-specific)
IF NOT permStart.sts.bOK THEN
    Start := E_RpcMethodResponse.REJECTED_PERMISSIVE_NOT_MET;
    RETURN;
END_IF;

// Permission check (global auto permissives)
IF NOT permAuto.sts.bOK THEN
    Start := E_RpcMethodResponse.REJECTED_PERMISSIVE_NOT_MET;
    RETURN;
END_IF;

// Execute
_abortRequested := FALSE;
_pauseRequested := FALSE;
_homeRequested := FALSE;
_proceedRequested := FALSE;
_stopRequested := FALSE;
_completeStateRequested := FALSE;
_startRequested := TRUE;
Start := E_RpcMethodResponse.ACCEPTED;
END_METHOD

{attribute 'TcRpcEnable' := '1'}
METHOD Stop : E_RpcMethodResponse
VAR_INPUT
    eRequester : E_Requester := E_Requester.PROG;
END_VAR
// Safety command - skip source check, skip fault check
IF Status.State = E_SM_State.STOPPED OR Status.State = E_SM_State.STOPPING THEN
    Stop := E_RpcMethodResponse.REJECTED_WRONG_STATE;
    RETURN;
END_IF;

// Execute
_abortRequested := FALSE;
_homeRequested := FALSE;
_proceedRequested := FALSE;
_startRequested := FALSE;
_pauseRequested := FALSE;
_completeStateRequested := FALSE;
_stopRequested := TRUE;
Stop := E_RpcMethodResponse.ACCEPTED;
END_METHOD

{attribute 'TcRpcEnable' := '1'}
// Map a running interlock bit. Call every cycle. bGood=TRUE means the condition is safe.
// If bGood goes FALSE from any non-stopped state the machine auto-aborts.
METHOD MapRunningIntlk
VAR_INPUT
    bitIndex : UDINT;
    bGood    : BOOL;
END_VAR
intlkRunning.MapInput(bitIndex := bitIndex, inputValue := bGood);
END_METHOD

{attribute 'TcRpcEnable' := '1'}
// Clear latched running interlock bits after the real-world condition has recovered.
// The machine will still be in STOPPED/ABORTING — issue Home/Start separately.
METHOD ResetRunningIntlk
intlkRunning.Reset();
END_METHOD

// INTERNAL: used by FB_Step to advance the sequence. Not part of the user API.
METHOD INTERNAL SetNextStep
VAR_INPUT
    nStep : DINT;
END_VAR
_nextStep := nStep;
END_METHOD

// INTERNAL: used by FB_Step to publish its name to StepInfo. Not part of the user API.
METHOD INTERNAL SetStepName
VAR_INPUT
    sName : STRING(40);
END_VAR
Status.Step.Name := sName;
END_METHOD

// INTERNAL: used by FB_Step to publish the active step permissive data for HMI / OPC.
METHOD INTERNAL SetStepPermissives
VAR_INPUT
        cfg : ST_Permissive_Config;
        sts : ST_Permissive_Status;
END_VAR
Status.Step.PermCfg := cfg;
Status.Step.PermStatus := sts;
END_METHOD

// INTERNAL: used by FB_Step to fault the current step (timeout, etc.).
// Faults by advancing to the next (odd) step number -- Status.Faulted derives
// from (CurrentStep MOD 2). Not part of the user API.
METHOD INTERNAL SetStepFault
VAR_INPUT
    bFault : BOOL;
END_VAR
IF bFault THEN
    _nextStep := Status.Step.Current + 1;
END_IF;
END_METHOD

END_FUNCTION_BLOCK

// ---- Modules/Sequencing/StateMachine/FB_Step.TcPOU
(*
FB_Step - Lightweight step lifecycle wrapper
============================================
Each step in a sequence is one FB_Step instance. The parent FB_StateMachine
owns the active step number, step timer, fault detection, and command handling.
This FB only reports "am I active?" and drives the Entry/Execute/Exit/Advance
lifecycle for the user's code.

Lifecycle (while this step is the SM's active step):
  Entry   : TRUE one scan on activation         -> one-shot init
  Execute : TRUE every scan until perms satisfied -> cyclic work + MapPerm
  Exiting : TRUE one scan after perms satisfied  -> one-shot cleanup
  Advance : writes nNextStep to the SM, SM increments on next scan

Branching / looping / jumping:
  nNextStep is a VAR_INPUT re-evaluated every scan. To branch, loop, or jump,
  just assign nNextStep dynamically in the call. There is no separate override
  method -- the input IS the dynamic target.

      step(sm := sm, nStep := 3004,
           nNextStep := SEL(bPass, 3500, 3006),  // branch inline
           nTimeout := 12, sName := 'Inspect');

  nNextStep := 0   -> completes the sequence (SM transitions to waiting state)
  nNextStep := N   -> SM advances to step N (any valid step; forward/back)

Note: 'Exiting' is used instead of 'Exit' because EXIT is an IEC reserved word.
*)
FUNCTION_BLOCK FB_Step
VAR_IN_OUT
    sm : FB_StateMachine;
END_VAR

VAR_INPUT
    nStep : DINT;
    nNextStep : DINT;
    nTimeout : DINT;
    sName : STRING(40);
END_VAR

VAR_OUTPUT
    Entry : BOOL;
    Execute : BOOL;
    Exiting : BOOL;
END_VAR

VAR
    _perms : FB_Permissives;
    _active : BOOL;
    _prevActive : BOOL;
    _permsSatisfied : BOOL;
    _permsEvalReady : BOOL;
    _exitDone : BOOL;
END_VAR


// Evaluate permissives (unmapped bits automatically good)
_perms();
_permsSatisfied := _perms.sts.bOK;

// Check if this step is the active step in the state machine
_active := (sm.Status.Step.Current = nStep);

// Reset lifecycle outputs each scan
Entry := FALSE;
Execute := FALSE;
Exiting := FALSE;

IF _active THEN
    // Publish step name to SM for HMI / diagnostics
    sm.SetStepName(sName);
  sm.SetStepPermissives(cfg := _perms.cfg, sts := _perms.sts);

    IF NOT _prevActive THEN
        //---------------------------------------------------------------------
        // ENTRY: first scan this step is active
        //---------------------------------------------------------------------
        Entry := TRUE;
        _permsEvalReady := FALSE;
        _exitDone := FALSE;

    ELSIF NOT _permsEvalReady THEN
        //---------------------------------------------------------------------
        // First EXECUTE scan: user is mapping perms this scan; evaluate next
        // scan so the first evaluation sees all MapPerm calls from this cycle.
        //---------------------------------------------------------------------
        Execute := TRUE;
        _permsEvalReady := TRUE;

    ELSIF NOT _permsSatisfied THEN
        //---------------------------------------------------------------------
        // EXECUTE: waiting for all mapped permissives to be satisfied
        //---------------------------------------------------------------------
        IF NOT sm.Status.Faulted THEN
            Execute := TRUE;
        END_IF;

        // Timeout fault detection
        IF nTimeout > 0 AND sm.Status.Step.TimerSeconds > DINT_TO_REAL(nTimeout) THEN
            sm.SetStepFault(bFault := TRUE);
        END_IF;

    ELSIF NOT _exitDone THEN
        //---------------------------------------------------------------------
        // EXIT: all permissives satisfied, one-scan cleanup
        //---------------------------------------------------------------------
        Exiting := TRUE;
        _exitDone := TRUE;

    ELSE
        //---------------------------------------------------------------------
        // ADVANCE: post-exit, hand the (current-scan) nNextStep to the SM.
        // Because nNextStep is re-evaluated every scan, the user's latest
        // branch decision wins -- no override method needed.
        //---------------------------------------------------------------------
        sm.SetNextStep(nStep := nNextStep);
    END_IF;

ELSE
    // Reset lifecycle tracking when step is not active
    _permsEvalReady := FALSE;
    _exitDone := FALSE;
END_IF;

_prevActive := _active;

METHOD MapPerm
VAR_INPUT
    nIndex : UDINT;
    sDescription : STRING;
    bValue : BOOL;
END_VAR
_perms.MapInput(bitIndex := nIndex, inputValue := bValue);
_perms.cfg.aNames[nIndex] := sDescription;
END_METHOD

END_FUNCTION_BLOCK
